RoboDK station: Example.rdk

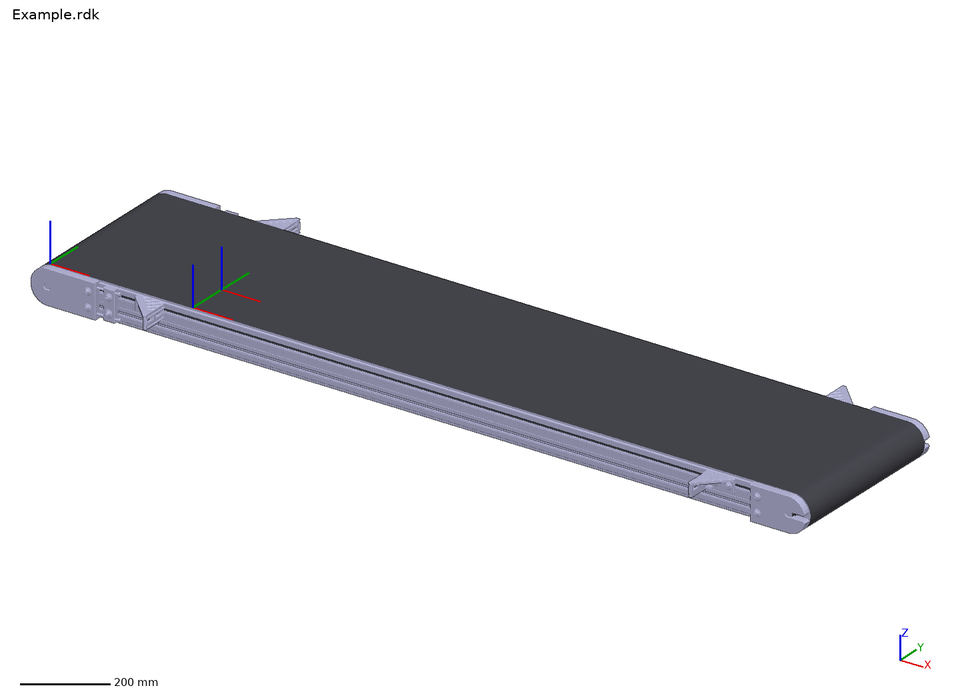
[picture v0: the station drawn from its stored meshes, robots at their saved joint values, targets as dots, program paths as lines]
Station Example (saved by RoboDK 5.3.2). Poses are relative to the parent item; angles as X-Y-Z fixed-axis rotations.
Station parameters (name, value as stored): Use Metric, True, BOXSPAWNER_SIZE_X, 150.0, BOXSPAWNER_SIZE_Y, 200.0, BOXSPAWNER_SIZE_Z, 250.0, BOXSPAWNER_UNITS, True, BOXSPAWNER_PARENT, Spawn Location, BOXSPAWNER_CONV_PARENT, Conveyor Frame
  - frame Conveyor Belt Base at (1150, 1000, 0) mm
    - robot Conveyor Belt: 1 axes
        modified DH rows (alpha deg, a mm, theta deg, d mm): 0, 0, 0, 0 linear
        base shift (0, 0, 0) mm, rotated rx 0 ry 90 rz 0 deg
        joint limits [-500000] to [500000]; home [0]; saved at [385]
      - frame Conveyor Frame at (0, 0, 0) mm
    - frame Spawn Location at (385, 110, 0) mm
  - Python program Spawn Box (listed below)

--- Python program Spawn Box ---
# Type help("robolink") or help("robodk") for more information
# Press F5 to run the script
# Documentation: https://robodk.com/doc/en/RoboDK-API.html
# Reference:     https://robodk.com/doc/en/PythonAPI/index.html
# Note: It is not required to keep a copy of this file, your python script is saved with the station
from robolink import Robolink  # RoboDK API
import SpawnBoxTools as spt

RDK = Robolink()
spt.loadParameters(RDK)
spt.createBox(RDK)
